% RSLogix 500 project LAB04_BAK006.RSS, saved by version 8.30.00.16 %
PROJECT "LAB4"    % processor: Bul.1763 MicroLogix 1100 Series B %

PROGRAM FILES
  LAD 2   3 rungs

DATA FILES
  O0 OUTPUT  4 elements
  I1 INPUT  6 elements
  S2 STATUS  66 elements
  B3 BINARY  1 elements
  T4 TIMER  1 elements
  C5 COUNTER  1 elements
  R6 CONTROL  1 elements
  N7 INTEGER  1 elements
  F8 FLOAT  1 elements

LADDER 2
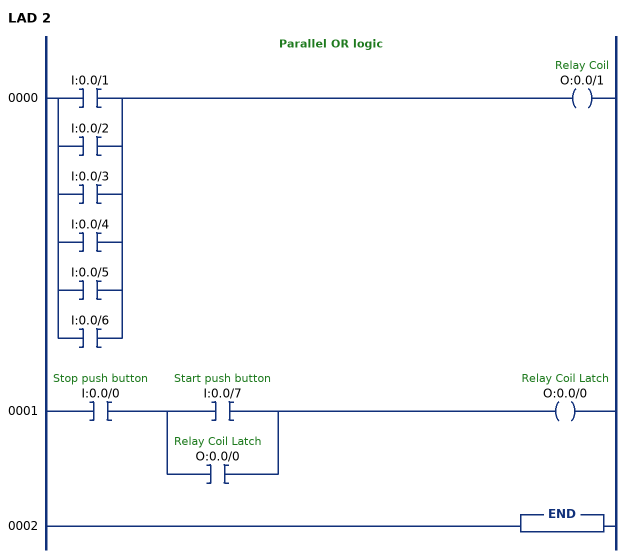
% Rung: 0 %
% TITLE: Parallel OR logic %
SOR BST XIC I:0.0/1 NXB XIC I:0.0/2 NXB XIC I:0.0/3 NXB XIC I:0.0/4 NXB XIC I:0.0/5 NXB XIC I:0.0/6 BND OTE O:0.0/1 EOR
%   O:0.0/1  "Relay Coil" %
% Rung: 1 %
SOR XIC I:0.0/0 BST XIC I:0.0/7 NXB XIC O:0.0/0 BND OTE O:0.0/0 EOR
%   I:0.0/0  "Stop push button" %
%   I:0.0/7  "Start push button" %
%   O:0.0/0  "Relay Coil Latch" %
% Rung: 2 %
SOR END EOR
